TYPE ST_MC_CMD :
STRUCT
	bExe			:BOOL;
	lrVelocity		:LREAL;
	lrAcceleration 	:LREAL;
	lrDeceleration 	:LREAL;
	lrJerk		 	:LREAL;
	lrDistance	 	:LREAL;
	lrPosition	 	:LREAL;
	EnuDirection	:MC_Direction;
	EnuBufferMode	:MC_BufferMode;
	EnuOptions		:ST_MoveOptions;
	
	
END_STRUCT
END_TYPE

(* stored: Version 1.1.0.1, ProductVersion 3.1.4024.9
   DUT ST_MC_CMD: Id {dee0747b-e8df-40c1-a827-038bbdedd45b} *)
